FUNCTION_BLOCK Test_F_TimeAsString_ReturnsTimeStringWithLeadingZeros EXTENDS T_UnitTestBase
VAR
    TimeStruct : TIMESTRUCT := (wHour := 6, wMinute := 5, wSecond := 4);
END_VAR

Assertion.AssertEquals_STRING(
    Expected := '06:05:04',
    Actual   := F_TimeAsString(TimeStruct),
    VariableName  := 'F_TimeAsString(TimeStruct)');


TestFinished();

END_FUNCTION_BLOCK

(* stored: Version 1.1.0.1, ProductVersion 3.1.4024.4
   POU Test_F_TimeAsString_ReturnsTimeStringWithLeadingZeros: Id {72a01420-e5e9-02f9-2a71-637672ec7977}, SpecialFunc None *)
